{attribute 'TcDependOnClassFactory' := 'WeldingArm6AxisMotion_Control'}
FUNCTION_BLOCK FB_WeldingArm6AxisMotion_Control EXTENDS FB_TcMatSimObject
VAR_INPUT
	stInput: ST_WeldingArm6AxisMotion_Control_Input;
END_VAR
VAR_OUTPUT
	stOutput: ST_WeldingArm6AxisMotion_Control_Output;
END_VAR
VAR
	stInitData: ST_WeldingArm6AxisMotion_Control_InitData;
	arrDataAreas: ARRAY[1..2] OF ST_TcMatSimObjectDataAreaInfo;
	bParametersVerified: BOOL;
END_VAR

PROPERTY CallBy_Online : TctModuleCallByType
GET
hResult := GetObjPara(16#00000000,sizeof(CallBy_Online),adr(CallBy_Online));
END_GET
SET
hResult := SetObjPara(16#00000000,sizeof(CallBy_Online),adr(CallBy_Online));
END_SET
END_PROPERTY

PROPERTY CallBy_Startup : TctModuleCallByType
GET
CallBy_Startup := stInitData.CallBy;
END_GET
SET
stInitData.CallBy := CallBy_Startup;
END_SET
END_PROPERTY

PROPERTY ContextInfoArr_0_TaskCycleTimeNs_Online : UDINT
GET
hResult := GetObjPara(16#03002080,sizeof(ContextInfoArr_0_TaskCycleTimeNs_Online),adr(ContextInfoArr_0_TaskCycleTimeNs_Online));
END_GET
SET
hResult := SetObjPara(16#03002080,sizeof(ContextInfoArr_0_TaskCycleTimeNs_Online),adr(ContextInfoArr_0_TaskCycleTimeNs_Online));
END_SET
END_PROPERTY

PROPERTY ContextInfoArr_0_TaskCycleTimeNs_Startup : UDINT
GET
ContextInfoArr_0_TaskCycleTimeNs_Startup := stInitData.ContextInfoArr_0_TaskCycleTimeNs;
END_GET
SET
stInitData.ContextInfoArr_0_TaskCycleTimeNs := ContextInfoArr_0_TaskCycleTimeNs_Startup;
END_SET
END_PROPERTY

PROPERTY ContextInfoArr_0_TaskOid_Online : OTCID
GET
hResult := GetObjPara(16#03002060,sizeof(ContextInfoArr_0_TaskOid_Online),adr(ContextInfoArr_0_TaskOid_Online));
END_GET
SET
hResult := SetObjPara(16#03002060,sizeof(ContextInfoArr_0_TaskOid_Online),adr(ContextInfoArr_0_TaskOid_Online));
END_SET
END_PROPERTY

PROPERTY ContextInfoArr_0_TaskOid_Startup : OTCID
GET
ContextInfoArr_0_TaskOid_Startup := stInitData.ContextInfoArr_0_TaskOid;
END_GET
SET
stInitData.ContextInfoArr_0_TaskOid := ContextInfoArr_0_TaskOid_Startup;
END_SET
END_PROPERTY

PROPERTY ContextInfoArr_0_TaskPort_Online : UINT
GET
hResult := GetObjPara(16#03002090,sizeof(ContextInfoArr_0_TaskPort_Online),adr(ContextInfoArr_0_TaskPort_Online));
END_GET
SET
hResult := SetObjPara(16#03002090,sizeof(ContextInfoArr_0_TaskPort_Online),adr(ContextInfoArr_0_TaskPort_Online));
END_SET
END_PROPERTY

PROPERTY ContextInfoArr_0_TaskPort_Startup : UINT
GET
ContextInfoArr_0_TaskPort_Startup := stInitData.ContextInfoArr_0_TaskPort;
END_GET
SET
stInitData.ContextInfoArr_0_TaskPort := ContextInfoArr_0_TaskPort_Startup;
END_SET
END_PROPERTY

PROPERTY ContextInfoArr_0_TaskPriority_Online : UDINT
GET
hResult := GetObjPara(16#03002070,sizeof(ContextInfoArr_0_TaskPriority_Online),adr(ContextInfoArr_0_TaskPriority_Online));
END_GET
SET
hResult := SetObjPara(16#03002070,sizeof(ContextInfoArr_0_TaskPriority_Online),adr(ContextInfoArr_0_TaskPriority_Online));
END_SET
END_PROPERTY

PROPERTY ContextInfoArr_0_TaskPriority_Startup : UDINT
GET
ContextInfoArr_0_TaskPriority_Startup := stInitData.ContextInfoArr_0_TaskPriority;
END_GET
SET
stInitData.ContextInfoArr_0_TaskPriority := ContextInfoArr_0_TaskPriority_Startup;
END_SET
END_PROPERTY

PROPERTY ContextInfoArr_0_TaskSortOrder_Online : UDINT
GET
hResult := GetObjPara(16#030020b0,sizeof(ContextInfoArr_0_TaskSortOrder_Online),adr(ContextInfoArr_0_TaskSortOrder_Online));
END_GET
SET
hResult := SetObjPara(16#030020b0,sizeof(ContextInfoArr_0_TaskSortOrder_Online),adr(ContextInfoArr_0_TaskSortOrder_Online));
END_SET
END_PROPERTY

PROPERTY ContextInfoArr_0_TaskSortOrder_Startup : UDINT
GET
ContextInfoArr_0_TaskSortOrder_Startup := stInitData.ContextInfoArr_0_TaskSortOrder;
END_GET
SET
stInitData.ContextInfoArr_0_TaskSortOrder := ContextInfoArr_0_TaskSortOrder_Startup;
END_SET
END_PROPERTY

PROPERTY CycleUpdateExecuted_Online : BOOL
GET
hResult := GetObjPara(16#00000004,sizeof(CycleUpdateExecuted_Online),adr(CycleUpdateExecuted_Online));
END_GET
SET
hResult := SetObjPara(16#00000004,sizeof(CycleUpdateExecuted_Online),adr(CycleUpdateExecuted_Online));
END_SET
END_PROPERTY

METHOD Execute : HRESULT

IF (SUCCEEDED(hResult)) THEN
  hResult := VerifyParameters();
END_IF

	// update DataArea information
SetDataAreaInfo(ADR(arrDataAreas),2);
	
	// call base method
Execute := SUPER^.Execute();
END_METHOD

PROPERTY ExecuteModelCode_Online : BOOL
GET
hResult := GetObjPara(16#00000008,sizeof(ExecuteModelCode_Online),adr(ExecuteModelCode_Online));
END_GET
SET
hResult := SetObjPara(16#00000008,sizeof(ExecuteModelCode_Online),adr(ExecuteModelCode_Online));
END_SET
END_PROPERTY

PROPERTY ExecuteModelCode_Startup : BOOL
GET
ExecuteModelCode_Startup := stInitData.ExecuteModelCode;
END_GET
SET
stInitData.ExecuteModelCode := ExecuteModelCode_Startup;
END_SET
END_PROPERTY

PROPERTY ExecutionSequence_Online : TctModuleExecutionSequenceType
GET
hResult := GetObjPara(16#00000001,sizeof(ExecutionSequence_Online),adr(ExecutionSequence_Online));
END_GET
SET
hResult := SetObjPara(16#00000001,sizeof(ExecutionSequence_Online),adr(ExecutionSequence_Online));
END_SET
END_PROPERTY

PROPERTY ExecutionSequence_Startup : TctModuleExecutionSequenceType
GET
ExecutionSequence_Startup := stInitData.ExecutionSequence;
END_GET
SET
stInitData.ExecutionSequence := ExecutionSequence_Startup;
END_SET
END_PROPERTY

METHOD FB_init : BOOL
VAR_INPUT
	/// if TRUE, the retain variables are initialized (warm start / cold start)
	bInitRetains: BOOL;
	/// if TRUE, the instance afterwards gets moved into the copy code (online change)
	bInCopyCode: BOOL;
	oid: OTCID;
END_VAR
VAR
	clsId: CLSID;
END_VAR

// initialize flags
bParametersVerified := false;
                    
// set module class id for compatibility check
clsId.Data1 := 16#412caec1;
clsId.Data2 := 16#7008;
clsId.Data3 := 16#47ed;
clsId.Data4[0] := 16#9b;
clsId.Data4[1] := 16#82;
clsId.Data4[2] := 16#ce;
clsId.Data4[3] := 16#15;
clsId.Data4[4] := 16#e3;
clsId.Data4[5] := 16#d3;
clsId.Data4[6] := 16#23;
clsId.Data4[7] := 16#f9;

AssignClassId(clsId);
                    
// initialize InitData structure with default values              
stInitData.CallByHdr.indexGroup := 0;
stInitData.CallByHdr.indexOffset := 16#00000000;
stInitData.CallByHdr.cbData := SIZEOF(stInitData.CallBy);
stInitData.CallBy := TctModuleCallByType.Module;
stInitData.ExecutionSequenceHdr.indexGroup := 0;
stInitData.ExecutionSequenceHdr.indexOffset := 16#00000001;
stInitData.ExecutionSequenceHdr.cbData := SIZEOF(stInitData.ExecutionSequence);
stInitData.ExecutionSequence := TctModuleExecutionSequenceType.StateUpdateAfterOutputMapping;
stInitData.StepSizeHdr.indexGroup := 0;
stInitData.StepSizeHdr.indexOffset := 16#00000002;
stInitData.StepSizeHdr.cbData := SIZEOF(stInitData.StepSize);
stInitData.StepSize := TctStepSizeType.UseTaskCycleTime;
stInitData.ExecuteModelCodeHdr.indexGroup := 0;
stInitData.ExecuteModelCodeHdr.indexOffset := 16#00000008;
stInitData.ExecuteModelCodeHdr.cbData := SIZEOF(stInitData.ExecuteModelCode);
stInitData.ExecuteModelCode := 1;
stInitData.ModelParametersHdr.indexGroup := 0;
stInitData.ModelParametersHdr.indexOffset := 16#82000000;
stInitData.ModelParametersHdr.cbData := SIZEOF(stInitData.ModelParameters);
stInitData.ModelParameters.tcycle_Value := 5.00000000000000000e+00;
stInitData.ModelParameters.J1rg_Value[0] := 2.00000000000000000e+01;
stInitData.ModelParameters.J1rg_Value[1] := 2.00000000000000000e+02;
stInitData.ModelParameters.J2rg_Value[0] := -2.70000000000000000e+02;
stInitData.ModelParameters.J2rg_Value[1] := 9.00000000000000000e+01;
stInitData.ModelParameters.J3rg_Value[0] := 2.00000000000000000e+01;
stInitData.ModelParameters.J3rg_Value[1] := 1.30000000000000000e+02;
stInitData.ModelParameters.phirg_Value[0] := -3.00000000000000000e+01;
stInitData.ModelParameters.phirg_Value[1] := 3.00000000000000000e+01;
stInitData.ModelParameters.gamarg_Value[0] := 1.50000000000000000e+01;
stInitData.ModelParameters.gamarg_Value[1] := 3.50000000000000000e+01;
stInitData.ContextInfoArr_0_TaskOidHdr.indexGroup := 0;
stInitData.ContextInfoArr_0_TaskOidHdr.indexOffset := 16#03002060;
stInitData.ContextInfoArr_0_TaskOidHdr.cbData := SIZEOF(stInitData.ContextInfoArr_0_TaskOid);
stInitData.ContextInfoArr_0_TaskPriorityHdr.indexGroup := 0;
stInitData.ContextInfoArr_0_TaskPriorityHdr.indexOffset := 16#03002070;
stInitData.ContextInfoArr_0_TaskPriorityHdr.cbData := SIZEOF(stInitData.ContextInfoArr_0_TaskPriority);
stInitData.ContextInfoArr_0_TaskCycleTimeNsHdr.indexGroup := 0;
stInitData.ContextInfoArr_0_TaskCycleTimeNsHdr.indexOffset := 16#03002080;
stInitData.ContextInfoArr_0_TaskCycleTimeNsHdr.cbData := SIZEOF(stInitData.ContextInfoArr_0_TaskCycleTimeNs);
stInitData.ContextInfoArr_0_TaskPortHdr.indexGroup := 0;
stInitData.ContextInfoArr_0_TaskPortHdr.indexOffset := 16#03002090;
stInitData.ContextInfoArr_0_TaskPortHdr.cbData := SIZEOF(stInitData.ContextInfoArr_0_TaskPort);
stInitData.ContextInfoArr_0_TaskSortOrderHdr.indexGroup := 0;
stInitData.ContextInfoArr_0_TaskSortOrderHdr.indexOffset := 16#030020b0;
stInitData.ContextInfoArr_0_TaskSortOrderHdr.cbData := SIZEOF(stInitData.ContextInfoArr_0_TaskSortOrder);
stInitData.Header.cbData := SIZEOF(stInitData)-SIZEOF(stInitData.Header);
stInitData.Header.uiElmCnt := 10;


// set pointer to InitData structure
SetInitDataInfo(ADR(stInitData));

// set DataArea information
SetDataAreaInfo(ADR(arrDataAreas),2);
arrDataAreas[1].nDataAreaId := 0;
arrDataAreas[1].nSize := SIZEOF(stInput);
arrDataAreas[1].pPlcVar := ADR(stInput);
arrDataAreas[1].pModuleProcImg := 0;
arrDataAreas[1].eDataAreaType := E_TcMatSimDataAreaType.InputDst;
arrDataAreas[2].nDataAreaId := 1;
arrDataAreas[2].nSize := SIZEOF(stOutput);
arrDataAreas[2].pPlcVar := ADR(stOutput);
arrDataAreas[2].pModuleProcImg := 0;
arrDataAreas[2].eDataAreaType := E_TcMatSimDataAreaType.OutputSrc;


// initialize basic interface pointers and return
FB_init := SUCCEEDED(Init(oid));
END_METHOD

PROPERTY InitData : ST_WeldingArm6AxisMotion_Control_InitData
GET
InitData := stInitData;
END_GET
SET
stInitData := InitData;
END_SET
END_PROPERTY

PROPERTY Input_Online : ExtU_weldingArm6axisMotionTes_T
GET
hResult := GetObjPara(16#80000000,sizeof(Input_Online),adr(Input_Online));
END_GET
SET
hResult := SetObjPara(16#80000000,sizeof(Input_Online),adr(Input_Online));
END_SET
END_PROPERTY

{attribute 'object_name' := 'Internal_SetObjState'}
METHOD PROTECTED Internal_SetObjState
VAR_INPUT
	hr: REFERENCE TO HRESULT;
	nextState: TCOM_STATE;
END_VAR

// update pointer to InitData structure
SetInitDataInfo(ADR(stInitData));
// call base method
SUPER^.Internal_SetObjState(hr,nextState);
END_METHOD

PROPERTY MdlInitialized_Online : BOOL
GET
hResult := GetObjPara(16#00000003,sizeof(MdlInitialized_Online),adr(MdlInitialized_Online));
END_GET
SET
hResult := SetObjPara(16#00000003,sizeof(MdlInitialized_Online),adr(MdlInitialized_Online));
END_SET
END_PROPERTY

PROPERTY ModelParameters_Online : P_weldingArm6axisMotionTest1_T
GET
hResult := GetObjPara(16#82000000,sizeof(ModelParameters_Online),adr(ModelParameters_Online));
END_GET
SET
hResult := SetObjPara(16#82000000,sizeof(ModelParameters_Online),adr(ModelParameters_Online));
END_SET
END_PROPERTY

PROPERTY ModelParameters_Startup : P_weldingArm6axisMotionTest1_T
GET
ModelParameters_Startup := stInitData.ModelParameters;
END_GET
SET
stInitData.ModelParameters := ModelParameters_Startup;
END_SET
END_PROPERTY

PROPERTY ModuleBuildInfo_Online : TctModuleBuildInfoType
GET
hResult := GetObjPara(16#00000007,sizeof(ModuleBuildInfo_Online),adr(ModuleBuildInfo_Online));
END_GET
SET
hResult := SetObjPara(16#00000007,sizeof(ModuleBuildInfo_Online),adr(ModuleBuildInfo_Online));
END_SET
END_PROPERTY

PROPERTY ModuleInfo_Online : TctModuleInfoType
GET
hResult := GetObjPara(16#00000006,sizeof(ModuleInfo_Online),adr(ModuleInfo_Online));
END_GET
SET
hResult := SetObjPara(16#00000006,sizeof(ModuleInfo_Online),adr(ModuleInfo_Online));
END_SET
END_PROPERTY

{attribute 'object_name' := 'SaveOnlineParametersForInit'}
METHOD SaveOnlineParametersForInit : HRESULT
VAR
	idx: UINT;
	pInitElemHdr: POINTER TO TComInitDataElmHdr;
	pData: PVOID;
	nData: UDINT;
END_VAR
VAR CONSTANT
	nInitDataAlignment: UDINT := 4;
END_VAR

// update pointer to InitData structure
SetInitDataInfo(ADR(stInitData));
// call base method
SaveOnlineParametersForInit := SUPER^.SaveOnlineParametersForInit();
END_METHOD

PROPERTY SimulinkTime_Online : LREAL
GET
hResult := GetObjPara(16#00000005,sizeof(SimulinkTime_Online),adr(SimulinkTime_Online));
END_GET
SET
hResult := SetObjPara(16#00000005,sizeof(SimulinkTime_Online),adr(SimulinkTime_Online));
END_SET
END_PROPERTY

PROPERTY StepSize_Online : TctStepSizeType
GET
hResult := GetObjPara(16#00000002,sizeof(StepSize_Online),adr(StepSize_Online));
END_GET
SET
hResult := SetObjPara(16#00000002,sizeof(StepSize_Online),adr(StepSize_Online));
END_SET
END_PROPERTY

PROPERTY StepSize_Startup : TctStepSizeType
GET
StepSize_Startup := stInitData.StepSize;
END_GET
SET
stInitData.StepSize := StepSize_Startup;
END_SET
END_PROPERTY

{attribute 'object_name' := 'VerifyParameters'}
METHOD PRIVATE VerifyParameters : HRESULT
VAR
	moduleCallByParam: TctModuleCallByType;
END_VAR

IF (bParametersVerified) THEN
  VerifyParameters := Tc2_System.E_HRESULTAdsErr.HRESULT_ADS_NOERROR;
ELSE
  VerifyParameters := GetObjPara(stInitData.CallByHdr.indexOffset,SIZEOF(moduleCallByParam),ADR(moduleCallByParam));
  
  // check the "CallBy" parameter to be set to "Module"
  IF (SUCCEEDED(VerifyParameters) AND (moduleCallByParam <> TctModuleCallByType.Module)) THEN
      VerifyParameters := Tc2_System.E_HRESULTAdsErr.INVALIDPARM;
  END_IF
  
  // set the parameters verified flag
  bParametersVerified := SUCCEEDED(VerifyParameters);
END_IF
END_METHOD

END_FUNCTION_BLOCK

(* stored: Version 1.1.0.1, ProductVersion 3.1.4020.12
   POU FB_WeldingArm6AxisMotion_Control: Id {72d8e695-881f-4689-b43e-43dcc8462e5d}, SpecialFunc None
   Property CallBy_Online: Id {f6a3d72c-9021-47bc-b838-e7c7d03832eb}
   Get Get: Id {f2aa0b5c-a703-4335-b601-3d64b7876896}
   Set Set: Id {7b5b9b93-0625-48aa-a1e0-f7162399a5e7}
   Property CallBy_Startup: Id {52fe5a66-e6ef-4215-ad6c-f202d937bb48}
   Get Get: Id {c6eb1260-1c4d-4258-8cfa-f1b70a9c55a9}
   Set Set: Id {0050a658-a701-4aae-aec4-2c46b0c9f37e}
   Property ContextInfoArr_0_TaskCycleTimeNs_Online: Id {5bfad9e2-9f82-4367-b10c-bb7f9aad45d8}
   Get Get: Id {fb16f9e5-291e-4775-a953-ea185710d66b}
   Set Set: Id {a2bd84c3-84b1-4221-9fcc-f3daa1f0c3c3}
   Property ContextInfoArr_0_TaskCycleTimeNs_Startup: Id {32aba032-398f-47d9-a97f-1e3862159f30}
   Get Get: Id {a115ac0c-b97d-42a3-8973-fb63dbb8db39}
   Set Set: Id {f0a661d8-05e7-4d6b-bb2f-444981ecd284}
   Property ContextInfoArr_0_TaskOid_Online: Id {15267122-435b-4d6f-9b94-275e11dfc7b2}
   Get Get: Id {11f3add4-a145-4766-b019-74d97b56e048}
   Set Set: Id {8086bc06-ee9b-4884-bed1-756036b98106}
   Property ContextInfoArr_0_TaskOid_Startup: Id {c9bea4dd-d1a5-4456-b7e2-be72db62d9c0}
   Get Get: Id {23240695-77b0-4330-8aa0-7e8ce3ef2f66}
   Set Set: Id {f80c44d5-5cd9-43c2-8f56-04914e6e54e3}
   Property ContextInfoArr_0_TaskPort_Online: Id {074bf85a-c7fb-43cf-96ea-863f7106946a}
   Get Get: Id {c3eb02d0-f853-4b28-a516-41d7632b32eb}
   Set Set: Id {c1175061-d92a-4226-bcda-98626c3e5dce}
   Property ContextInfoArr_0_TaskPort_Startup: Id {a855056c-4879-4b43-b03f-cf7f7d589d9b}
   Get Get: Id {3213c06f-cfec-4c43-afe0-7bb66ba8e452}
   Set Set: Id {aa034252-c665-4dfe-ae28-14bd051f8c3d}
   Property ContextInfoArr_0_TaskPriority_Online: Id {4db75e76-029d-4073-b26e-80408b98f974}
   Get Get: Id {953a29a4-15e7-4f4a-b915-150bbd76e89a}
   Set Set: Id {5149640a-53e7-4a10-a8a6-ba6710404de7}
   Property ContextInfoArr_0_TaskPriority_Startup: Id {87283cb7-d278-424b-b0d4-ad617c10b85e}
   Get Get: Id {776b76e7-eef9-4878-91c8-2eba5a6298d7}
   Set Set: Id {cd6ad851-cc4a-4777-a2d7-694668011bdb}
   Property ContextInfoArr_0_TaskSortOrder_Online: Id {9deca592-a2e8-4049-b417-2d2c086710e3}
   Get Get: Id {fbee8046-39f7-4d35-ba23-0162d495e061}
   Set Set: Id {6139096d-c80b-407a-82cf-471f9a9204b2}
   Property ContextInfoArr_0_TaskSortOrder_Startup: Id {06ee9178-88b2-46d3-82e8-f132658f0860}
   Get Get: Id {0b71e846-8dc0-489e-b0b9-81252e5608b2}
   Set Set: Id {de397ac5-ff80-406e-b048-0b4002186e8e}
   Property CycleUpdateExecuted_Online: Id {4e38b47d-d9e9-4c35-8675-f5e6b9012c3f}
   Get Get: Id {7b721ce0-2064-4d06-aae9-e56a48e97daa}
   Set Set: Id {a3640c53-f33a-4e8a-b1d4-7dfaaa85a933}
   Method Execute: Id {0aac5514-388a-48b5-9ca5-cd3ea6b8fe48}
   Property ExecuteModelCode_Online: Id {836b432b-6fb8-44a1-8b72-cee1134cbb49}
   Get Get: Id {b42f41fb-43a3-4929-9ba1-7109f4ba0074}
   Set Set: Id {54a8716e-7efb-4b2e-bb5f-605a738cb358}
   Property ExecuteModelCode_Startup: Id {2297bec1-0c91-479e-9440-eafcf16a1acc}
   Get Get: Id {b1d909a1-522b-4aad-ae23-751aed22c0d6}
   Set Set: Id {591cb88c-1434-40ab-856b-e48fd3413b67}
   Property ExecutionSequence_Online: Id {8e2944d7-31c4-4161-bf84-610a0f528293}
   Get Get: Id {87593c5b-14d6-4b02-87df-21265c5d54f1}
   Set Set: Id {90e14c3c-9467-4bda-afc6-85077f13f334}
   Property ExecutionSequence_Startup: Id {01bc8908-ec67-4e03-8fda-fe58b5605235}
   Get Get: Id {50afaa7a-2109-4dc8-b742-5010bf9e085f}
   Set Set: Id {25a175ae-b8f9-44e6-b9f5-002e0cdc67c0}
   Method FB_init: Id {ef1e3c45-5797-4934-880c-e23d9e751a63}
   Property InitData: Id {50905e7b-95b3-4e6a-add1-97dab8da02eb}
   Get Get: Id {8ae1d73d-7e47-401b-8d85-1f141ecbb62b}
   Set Set: Id {92d19e08-688c-4a4a-a39c-b4f6a265ebf4}
   Property Input_Online: Id {9f3196e9-a837-42ac-a095-1b2aa7caed12}
   Get Get: Id {c019ec8d-966e-42e4-9771-71c74fb120d2}
   Set Set: Id {6395b596-5ef6-45fb-858a-4bdf01c1fd3e}
   Method Internal_SetObjState: Id {1f12df60-cb2b-4121-8810-85bff5c8d581}
   Property MdlInitialized_Online: Id {0a289389-6c8c-4e68-8767-def7461fabea}
   Get Get: Id {36204974-692a-42a1-9939-1bafb5f80d30}
   Set Set: Id {7e051857-4d9d-46d4-97b3-eb4e1ff9b4ec}
   Property ModelParameters_Online: Id {b872656b-a7ff-4906-a512-ac6898816a2d}
   Get Get: Id {f282e386-520e-453b-a9ff-45b8c1cc4da6}
   Set Set: Id {e1376f1d-5585-4e5f-8d7e-f98551de93a0}
   Property ModelParameters_Startup: Id {efa4c257-879f-4d6e-a525-77b3f2469dac}
   Get Get: Id {bc4a97b7-879c-4f85-8307-d35baebc417c}
   Set Set: Id {ef848971-1e63-4498-a9b9-687f2ff43cb5}
   Property ModuleBuildInfo_Online: Id {dbbd786d-c6b7-4498-886a-300ec41ead88}
   Get Get: Id {0f902d45-fd17-49c4-ae35-96d2f5eaced1}
   Set Set: Id {4265d731-e0ad-4afe-81dd-75e154a26477}
   Property ModuleInfo_Online: Id {0ca0b693-a39a-4ebc-aec6-24f1bf065362}
   Get Get: Id {5cdacd9e-1d1e-46b2-b049-738f91ac16e2}
   Set Set: Id {e985d8d2-8c4d-405a-80a1-067b66735b4a}
   Method SaveOnlineParametersForInit: Id {ae55b35c-8c74-46ba-9e31-16a257cfbb14}
   Property SimulinkTime_Online: Id {1479ddd7-d519-410a-85bf-9e281e5654dd}
   Get Get: Id {b1f74ffd-9152-406e-8072-129850c1f661}
   Set Set: Id {f820684a-c792-4960-8293-c356bae38e8a}
   Property StepSize_Online: Id {ea31de27-b9f2-4d14-8f90-cbfd1c2c33a8}
   Get Get: Id {05646e51-acec-4dea-96f9-08cdf3e2ee28}
   Set Set: Id {e8176a50-826b-4c7b-b491-ea0bf885084a}
   Property StepSize_Startup: Id {034395d9-a4c1-4379-8fa8-e3a5121aea8a}
   Get Get: Id {8cfab0cb-f993-48b1-900e-147f547b3d8d}
   Set Set: Id {9e8f6c95-58bc-40dc-8703-12020d28b0f9}
   Method VerifyParameters: Id {ecfcefd3-05df-4f7c-94f1-18eedd4c38a7} *)
